Fanuc KAREL source: ko00080.KL

-- PROVISIONAL review KL for V770-1; original PC SHA256 7236c0b48bbe2e8d3eaa716ad3ce866db6ef3611e54a02b954f7c1c8dde2d4f1
-- Incomplete behavior may be omitted. Consult companion uncertainty JSON. Do not deploy.
PROGRAM KO00080
%NOLOCKGROUP
BEGIN
  -- UNRESOLVED_PC offsets 5-12; opcodes 9D,23
  -- UNRESOLVED_PC offsets 17-66; opcodes 27,22,1C,27,49,7E,AD,22,31,7E,4A
  -- UNRESOLVED_PC offsets 71-75; opcodes 7F
END KO00080
